// TIA Portal V20 export
ORGANIZATION_BLOCK "Main"   // OB1, LAD, ProgramCycle
// stored: AutoNumber false
BEGIN

REGION Network 1
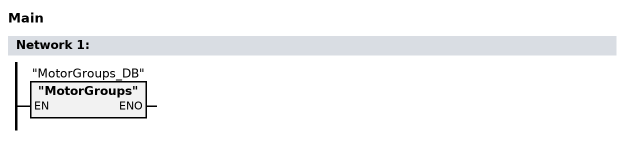
   RUNG wire#powerrail
      "MotorGroups_DB"()
   END_RUNG
   // the same network as SCL:
   "MotorGroups_DB"();   // "MotorGroups"
END_REGION
END_ORGANIZATION_BLOCK
